TYPE (* A Template for a Data Type *)
  (* Version 1.0, 2024-02-21, franz *)
  st8bits : STRUCT
    b0 : BOOL; (* BIT 00 *)
    b1 : BOOL; (* BIT 01 *)
    b2 : BOOL; (* BIT 02 *)
    b3 : BOOL; (* BIT 03 *)
    b4 : BOOL; (* BIT 04 *)
    b5 : BOOL; (* BIT 05 *)
    b6 : BOOL; (* BIT 06 *)
    b7 : BOOL; (* BIT 07 *)
  END_STRUCT;
END_TYPE
